// TIA Portal V17 export
// export: Created 2023-04-03T06:31:31.4738784Z, ExportSetting WithDefaults, DisplayName Totally Integrated Automation Portal, DisplayVersion V17 Update 4, DisplayName TIA Portal Openness, DisplayVersion V17 Update 4, DisplayName TIA Portal Version Control Interface, DisplayVersion V17, DisplayName STEP 7 Professional, DisplayVersion V17 Update 4, DisplayName STEP 7 Safety, DisplayVersion V17, DisplayName WinCC Professional, DisplayVersion V17 Update 4
DATA_BLOCK "ED"   // DB400
{ S7_Optimized_Access := 'TRUE' }
VERSION : 0.1
// stored: AutoNumber false, DBAccessibleFromOPCUA true, DBAccessibleFromWebserver true, IsOnlyStoredInLoadMemory false, IsRetainMemResEnabled false, IsWriteProtectedInAS false, MemoryReserve 100
   VAR
      Pems : Struct
         LinkState : Array[1..52] of "LPNDR_typePortLinkState";
         X1 : Bool;
         X2 : Bool;
         X3 : Bool;
      END_STRUCT;
      ET200 : Struct
         LinkState : Array[1..52] of "LPNDR_typePortLinkState";
         X1 : Bool;
         X2 : Bool;
      END_STRUCT;
   END_VAR
BEGIN
END_DATA_BLOCK
